TYPE ST_ProfinetMasterConfig :
(* EL6631 *)
STRUCT
	strTAMSNETID_ProfinetMasterEthercatAmsNetId			: T_AmsNetId:=''; (* string(23) *)
	strIPAddress										: STRING(15) := ''; (* currently display only not linked *)

END_STRUCT
END_TYPE

(* stored: Version 1.1.0.1
   DUT ST_ProfinetMasterConfig: Id {6de4214a-eb9c-49b5-84c7-d67a3026d335} *)
